{attribute addProperty BoxType "EJ2521-0224-0016"}
{attribute addProperty Id "Frequency_selectBIT10.1251Disable_rampBIT10.1252Go_counterBIT10.1253"}
{attribute addProperty CRC "2716536400"}
{attribute addProperty SizeInBites "16"}
{attribute addProperty SizeInBytes "2"}
TYPE Control_A1EB0E50 :
STRUCT
	{attribute addProperty Name "Frequency_select"}
	Frequency_select : BOOL;
	{attribute addProperty Name "Disable_ramp"}
	Disable_ramp : BOOL;
	{attribute addProperty Name "Go_counter"}
	Go_counter : BOOL;
	{attribute 'hide'}
	reserve_1_BIT_0 : BOOL;
	{attribute 'hide'}
	reserve_1_BIT_1 : BOOL;
	{attribute 'hide'}
	reserve_1_BIT_2 : BOOL;
	{attribute 'hide'}
	reserve_1_BIT_3 : BOOL;
	{attribute 'hide'}
	reserve_1_BIT_4 : BOOL;
	{attribute 'hide'}
	reserve_2 : BYTE;
END_STRUCT
END_TYPE

(* stored: Version 1.2.0.0, ProductVersion 3.1.4024.9
   DUT Control_A1EB0E50: Id {2cef6865-a5b3-42eb-9f41-c34dd122cefa} *)
